Fanuc KAREL source: ks00024.KL

-- PROVISIONAL review KL for V940-1; original PC SHA256 68f09371f8556af7dae3c7702a70d48cdc2e0a4afaffe824202312e1ccd99b73
-- Incomplete behavior may be omitted. Consult companion uncertainty JSON. Do not deploy.
PROGRAM KS00024
%NOLOCKGROUP
VAR
  FLAG : BOOLEAN
  N : INTEGER
  STATUS : INTEGER
  PN : STRING[80]
  VN : STRING[80]
-- UNRESOLVED_DECL A type=001101
-- UNRESOLVED_DECL B type=001101
BEGIN
  -- V9_ZERO_TABLE_METADATA_HINT layout=0002_ascii; no indexed target words; source/name/runtime held
  -- UNRESOLVED_PC offsets 5-13; opcodes 3F,75
  -- UNRESOLVED_PC offsets 18-27; opcodes 3F,75
  -- UNRESOLVED_PC offsets 32-47; opcodes 22,22,30
  -- UNRESOLVED_PC offsets 52-56; opcodes 7F
END KS00024
